(* IEC 61131-3 sources: axftcmlib/src/Axis, 9 files *)

(* ---- Axis.st ---- *)
USING Simatic.Ax.IO.Input;
USING System.Timer;
USING Simatic.Ax.SimpleControlModules;

NAMESPACE Simatic.Ax.axftcmlib
    TYPE INTERNAL
        StatesHoming : (Idle, MoveOutOfSensor, FindReferenceSensor, Done) := Idle;
    END_TYPE

    TYPE INTERNAL
        StateMoveAbsolute : (Idle, Moving, Stopping, Done) := Idle;
    END_TYPE

    TYPE INTERNAL
        MotionMode : (Stopped, Homing, MoveAbsolute, MoveRelative, MoveVelocity);
    END_TYPE

    TYPE
        PlcOpenState : (Ready, Busy, Done, Error) := Ready;
    END_TYPE

    ///Class contains all functions necessary for realisng a motion axis
    ///The motor is used for "powering" the axis
    ///The encoder is needed to monitor the current position
    CLASS Axis
        IMPLEMENTS IAxis
        VAR PUBLIC
            Motor : IMotor;
            Encoder : IEncoder;
            ReferenceSwitch : IBinSignal;
        END_VAR
        VAR PROTECTED
            _stateHoming : StatesHoming;
            _stateMoveAbsolute : StateMoveAbsolute;
            _motionMode : MotionMode;
            _velocity : LREAL;
            _direction : Direction;
            _position : LINT;
            _distance : LINT;
            _plcOpenState : PlcOpenState;
            _done : BOOL;
            _isHomed : BOOL;
            _statusRefSwitch : BOOL;
        END_VAR

        ///Outputs the current status of the axis and executes the protected methods(must be called in every cicle)
        METHOD PUBLIC RunCyclic
            _statusRefSwitch := ReferenceSwitch.Q();
            CASE _motionMode OF
                MotionMode#Stopped:
                    _plcOpenState := PlcOpenState#Ready;
                    ;
                MotionMode#Homing:
                    _plcOpenState := PlcOpenState#Busy;
                    _done := THIS._homing(velocity := _velocity, direction := _direction);
                    IF _done THEN
                        _plcOpenState := PlcOpenState#Done;
                        _isHomed := TRUE;
                        _motionMode := MotionMode#Stopped;
                    END_IF;
                MotionMode#MoveAbsolute:
                    IF (NOT (_isHomed)) THEN
                        _plcOpenState := PlcOpenState#Error;
                        RETURN;
                    END_IF;
                    _plcOpenState := PlcOpenState#Busy;
                    _done := THIS._moveAbsolute(velocity := _velocity, posititon := _position);
                    IF _done THEN
                        _plcOpenState := PlcOpenState#Done;
                        _motionMode := MotionMode#Stopped;
                    END_IF;
                    ;
                MotionMode#MoveRelative:
                    IF (NOT (_isHomed)) THEN
                        _plcOpenState := PlcOpenState#Error;
                        RETURN;
                    END_IF;
                    _plcOpenState := PlcOpenState#Busy;
                    _done := THIS._moveRelative(velocity := _velocity, distance := _distance);
                    IF _done THEN
                        _plcOpenState := PlcOpenState#Done;
                        _motionMode := MotionMode#Stopped;
                    END_IF;
                    ;
                MotionMode#MoveVelocity:
                    _plcOpenState := PlcOpenState#Busy;
                    Motor.Move(_velocity, _direction);

            END_CASE;
        END_METHOD

        ///Moves axis with a velocity
        /// Has to be stopped manually with Halt()
        METHOD PUBLIC MoveVelocity
            VAR_INPUT
                velocity : LREAL;
                direction : Direction;
            END_VAR
            _velocity := velocity;
             _direction := direction;
            _motionMode := MotionMode#MoveVelocity;
        END_METHOD

        ///Moves axis to a new position based on the current position
        METHOD PUBLIC MoveRelative : BOOL
            VAR_INPUT
                velocity : LREAL;
                distance : LINT;
            END_VAR
            _velocity := velocity;
            _distance := distance;
            _motionMode := MotionMode#MoveRelative;
        END_METHOD

        ///Moves axis to a new position based on the default position
        ///homing the axis beforehand is needed to execute this function
        METHOD PUBLIC MoveAbsolute : BOOL
            VAR_INPUT
                velocity : LREAL;
                position : LINT;
            END_VAR
            _velocity := velocity;
            _position := position;
            _motionMode := MotionMode#MoveAbsolute;
        END_METHOD

        ///Moves axis to the default "homing" position (needed for moveAbsolute())
        METHOD PUBLIC Homing : BOOL
            VAR_INPUT
                velocity : LREAL;
                direction : Direction;
            END_VAR
            _velocity := velocity;
            _direction := direction;
            _motionMode := MotionMode#Homing;
        END_METHOD

        ///Homes axis without moving it into default position
        ///Sets position to given value
        METHOD PUBLIC Homing : BOOL
            VAR_INPUT
                Position : LINT;
            END_VAR
            Encoder.SetValue(value := Position);
            _stateHoming := StatesHoming#Done;
            _plcOpenState := PlcOpenState#Done;
            _isHomed := TRUE;
        END_METHOD

        ///Stops movement of the axis
        ///needs to be called manually for MoveVelocity()
        METHOD PUBLIC Halt
            Motor.Halt();
            _motionMode := MotionMode#Stopped;
            _plcOpenState := PlcOpenState#Done;
        END_METHOD
        ///Checks whether the axis is homed or not
        METHOD PUBLIC IsHomed : BOOL
            IsHomed := _isHomed;
        END_METHOD

       //Protected methods are executed by RunCyclic()

       ///Moves axis with a velocity
        /// Has to be stopped manually with Halt()
        METHOD PROTECTED _moveVelocity
            VAR_INPUT
                velocity : LREAL;
                direction : Direction;
            END_VAR
            Motor.Move(velocity, direction);
        END_METHOD

        ///Moves axis to a new position based on the current position
        METHOD PROTECTED _moveRelative : BOOL
            VAR_INPUT
                velocity : LREAL;
                distance : LINT;
            END_VAR
            _moveRelative := THIS._moveAbsolute(velocity := velocity, posititon := Encoder.GetValue() + distance);
        END_METHOD

        ///Moves axis to a new position based on the default position
        ///homing the axis beforehand is needed to execute this function
        METHOD PROTECTED _moveAbsolute : BOOL
            VAR_INPUT
                velocity : LREAL;
                posititon : LINT;
            END_VAR
            VAR_TEMP
                dir : Direction;
            END_VAR
            CASE _stateMoveAbsolute OF
                StateMoveAbsolute#Idle:
                    IF (posititon = Encoder.GetValue()) THEN
                        _stateMoveAbsolute := StateMoveAbsolute#Done;
                        _moveAbsolute := TRUE;
                        Motor.Halt();
                    ELSE
                        _stateMoveAbsolute := StateMoveAbsolute#Moving;
                        Motor.Move(velocity, dir);
                    END_IF;
                    StateMoveAbsolute#Moving:
                    dir := THIS.DecideDirection(enc := Encoder, setPoint := posititon);
                    Motor.Move(velocity, dir);
                    IF (Encoder.GetValue() = posititon) THEN
                        _stateMoveAbsolute := StateMoveAbsolute#Done;
                        Motor.Halt();
                    END_IF;
                    StateMoveAbsolute#Done:
                    _moveAbsolute := TRUE;
                    _stateMoveAbsolute := StateMoveAbsolute#Idle;
                    ;
            END_CASE;
        END_METHOD

        ///Homes axis without moving it into default position
        ///Sets position to given value
        METHOD PROTECTED _homing : BOOL
            VAR_INPUT
                velocity : LREAL;
                direction : Direction;
            END_VAR
            // Reference switch already reached
            // Move out from the Reference switch in opposit direction
            CASE _stateHoming OF
                StatesHoming#Idle:
                    _isHomed := FALSE;
                    IF (ReferenceSwitch.Q()) THEN
                        _stateHoming := StatesHoming#MoveOutOfSensor;
                    ELSE
                        _stateHoming := StatesHoming#FindReferenceSensor;
                    END_IF;
                StatesHoming#MoveOutOfSensor:
                    Motor.Move(direction := THIS._oppositDirection(direction := direction));
                    IF (ReferenceSwitch.QFal()) THEN
                        Motor.Halt();
                        _stateHoming := StatesHoming#FindReferenceSensor;
                    END_IF;
                StatesHoming#FindReferenceSensor:
                    Motor.Move(direction := direction);
                    IF (ReferenceSwitch.QRis()) THEN
                        Motor.Halt();
                        Encoder.SetValue(value := 0);
                        _stateHoming := StatesHoming#Done;
                    END_IF;
                StatesHoming#Done:
                    _homing := TRUE;
                    _stateHoming := StatesHoming#Idle;
            END_CASE;
            ;
        END_METHOD

        ///inverts the current direction
        METHOD PROTECTED _oppositDirection : Direction
            VAR_INPUT
                direction : Direction;
            END_VAR
            IF (direction = Direction#Forward) THEN
                _oppositDirection := Direction#Reverse;
            ELSE
                _oppositDirection := Direction#Forward;
            END_IF;
        END_METHOD

        ///decides the needed direction to reach setpoint
        METHOD PROTECTED DecideDirection : Direction
            VAR_INPUT
                enc : IEncoder;
                setpoint : LINT;
            END_VAR
            IF (setpoint >= enc.GetValue()) THEN
                DecideDirection := Direction#Forward;
            ELSE
                DecideDirection := Direction#Reverse;
            END_IF;
        END_METHOD

        ///Outputs current status of the PLC
        METHOD PUBLIC GetPlcOpenState : PlcOpenState
            GetPlcOpenState := _plcOpenState;
        END_METHOD
        ///Returns whether the axis is busy with a movement command
        METHOD PUBLIC IsRunning : BOOL
            IsRunning := _plcOpenState = PlcOpenstate#Busy;
        END_METHOD
    END_CLASS

END_NAMESPACE

(* ---- IAxis.st ---- *)
NAMESPACE Simatic.Ax.axftcmlib

    TYPE
        Direction : (Forward, Reverse, Undefined) := Forward;
    END_TYPE

    ///Interface for implementing an axis
    ///Contains basic functions needed for realising an axis
    INTERFACE IAxis
        ///Moves axis wit given velcity in a given direction
        METHOD MoveVelocity
            VAR_INPUT
                velocity : LREAL;
                direction : Direction;
            END_VAR
        END_METHOD
        ///Moves axis to destination based on current position
        METHOD MoveRelative : BOOL
            VAR_INPUT
                velocity : LREAL;
                distance : LINT;
            END_VAR
        END_METHOD
        ///Moves axis to a new position based on the default position
        METHOD MoveAbsolute : BOOL
            VAR_INPUT
                velocity : LREAL;
                position : LINT;
            END_VAR
        END_METHOD
        ///Stops axis
        METHOD Halt
        END_METHOD
        ///Moves axis into the default position
        METHOD Homing : BOOL
            VAR_INPUT
                velocity : LREAL;
                direction : Direction;
            END_VAR
        END_METHOD
        ///Resets current position to deafult value without actual movement
        METHOD Homing : BOOL
            VAR_INPUT
                Position : LINT;
            END_VAR
        END_METHOD
        ///Returns whether the defaultposition is set
        METHOD IsHomed : BOOL
        END_METHOD
        ///Returns whether the axis is busy with a movement command
        METHOD IsRunning : BOOL
        END_METHOD
    END_INTERFACE

END_NAMESPACE

(* ---- IMotor.st ---- *)
NAMESPACE Simatic.Ax.axftcmlib
    INTERFACE IMotor
        METHOD Move
            VAR_INPUT
                velocity : LREAL;
                direction : Direction;
            END_VAR
        END_METHOD
        METHOD Halt
        END_METHOD
    END_INTERFACE
END_NAMESPACE

(* ---- ITimeprovider.st ---- *)
USING Siemens.Simatic.S71500.Clocks;
NAMESPACE Simatic.Ax.axftcmlib

    INTERFACE ITimeprovider
        Method GetElapsedSeconds :LREAL
        END_METHOD
    END_INTERFACE

    CLASS TimeProvider Implements ITimeprovider

    VAR
     _measurement : RuntimeMeasurement;
     _timeOfOperations : LTIME;
    END_VAR

    METHOD PUBLIC GetElapsedSeconds : LREAL
            _timeOfOperations := _measurement.Stop();
            GetElapsedSeconds := _measurement.GetElapsedSeconds();//time passed in seconds
            _measurement.Start();
    END_METHOD

    END_CLASS

    CLASS TimeProviderMOCK_100ms_const Implements ITimeprovider

        VAR
         _measurement : RuntimeMeasurement;
         _timeOfOperations : LTIME;
        END_VAR

        METHOD PUBLIC GetElapsedSeconds : LREAL
              GetElapsedSeconds := 0.1;
        END_METHOD

        END_CLASS

END_NAMESPACE

(* ---- AxisBase.st ---- *)
USING Simatic.Ax.Commands;

NAMESPACE Simatic.Ax.axftcmlib.Motion

    CLASS INTERNAL ABSTRACT AxisBase IMPLEMENTS itfAxis
        VAR PROTECTED
            _AxisRef : REF_TO TO_Axis;
        END_VAR

        METHOD PROTECTED ABSTRACT MakeAxisAbstract END_METHOD

        METHOD PUBLIC Attach
            VAR_INPUT
                axis : REF_TO TO_Axis;
            END_VAR
            _AxisRef := axis;
        END_METHOD

        METHOD PROTECTED IsAttached : BOOL
            IsAttached := _AxisRef <> NULL;
        END_METHOD

        METHOD PUBLIC PowerOn
            _AxisRef^.isPowerdOn := TRUE;
        END_METHOD

        METHOD PUBLIC PowerOff
            _AxisRef^.isPowerdOn := FALSE;
        END_METHOD

    END_CLASS

END_NAMESPACE

(* ---- Motor.st ---- *)
USING Simatic.Ax.IO.Output;
USING Simatic.Ax.axftcmlib;

NAMESPACE Simatic.Ax.axftcmlib

    CLASS MotorFT
        IMPLEMENTS IMotor
        VAR PUBLIC
            Forward : IBinOutput;
            Reverse : IBinOutput;
        END_VAR
        VAR PROTECTED
        END_VAR
        METHOD PUBLIC Move
            VAR_INPUT
                velocity : LREAL;
                direction : Direction;
            END_VAR
            IF (direction = Direction#Forward) THEN
                Forward.SetOn();
                Reverse.SetOff();
            ELSE
                Reverse.SetOn();
                Forward.SetOff();
            END_IF;
            ;
        END_METHOD
        METHOD PUBLIC Halt
            Reverse.SetOff();
            Forward.SetOff();
            ;
        END_METHOD
    END_CLASS

END_NAMESPACE

(* ---- PLCOpentateGuard.st ---- *)
USING Simatic.Ax.StateFramework;
NAMESPACE Simatic.Ax.axftcmlib
    // CLASS PLCOpenstateGuard IMPLEMENTS IGuard

    //     VAR PUBLIC
    //         UsedAxis : REF_TO AXIS;
    //     END_VAR

    //     VAR
    //         CurrentState : PlcOpenState;
    //     END_VAR

    //     METHOD PUBLIC Check : BOOL
    //         CurrentState := UsedAxis^.GetPlcOpenState();
    //        IF CurrentState = PlcOpenState#DONE THEN
    //         Check := TRUE;
    //        ELSE
    //         Check := FALSE;
    //        END_IF;
    //     END_METHOD

    //     METHOD PUBLIC Reset
    //         ;
    //     END_METHOD

    // END_CLASS
    CLASS PLCOpenstateGuard IMPLEMENTS IGuard
        VAR PUBLIC
            Axis : REF_TO Axis;
        END_VAR

        METHOD PUBLIC Check : BOOL
            Check := (Axis^.GetPlcOpenState() = PlcOpenState#Done);
        END_METHOD

        METHOD PUBLIC Reset
            ;
        END_METHOD
    END_CLASS
END_NAMESPACE

(* ---- TimeBasedEncoder.st ---- *)
USING Simatic.Ax.SimpleControlModules;
USING Simatic.Ax.IO.Output;
USING Simatic.Ax.IO.Input;

USING System.Timer;

NAMESPACE Simatic.Ax.axftcmlib
    CLASS TimeBasedEncoder Implements IEncoder
        VAR PUBLIC
            Velocity : LREAL; // m/s
            EncoderAxis : IAxis;
            TimeProvider : ITimeprovider;
            //--------------------------
            RealPosition : LREAL;
        END_VAR

        VAR PROTECTED
            _position : LREAL; // mm
        END_VAR

        /// Reset encoder position to zero
        METHOD PUBLIC Reset
            _position := 0.0;
        END_METHOD

        /// Set encoder to specific position
        /// value : Position which is set
        METHOD PUBLIC SetValue
            VAR_INPUT
                value : LINT;
            END_VAR
            _position := TO_LREAL(value);
        END_METHOD

        /// Returns the actual encoder position
        /// Actual encoder position
        METHOD PUBLIC GetValue : LINT
            GetValue := TO_LINT(_position);
            RealPosition := _position;
        END_METHOD

        /// Evaluate encoder signals
        METHOD PUBLIC Evaluate
            VAR_TEMP
             ds : LREAL;
             dt : LREAL;
            END_VAR

            dt := TimeProvider.GetElapsedSeconds();//time passed in seconds
            ds := Velocity * dt;
            IF (EncoderAxis.IsRunning()) THEN //If Axis is running
                _position := _position + ds;
            END_IF;
        END_METHOD
        //=========================================================
        /// Returns if the encoder has moved
        /// Encoder has moved
        METHOD PUBLIC HasMoved : BOOL
            // HasMoved := _encoderHasMoved;
            // _encoderHasMoved := FALSE;
           ;
        END_METHOD

        /// Counts the relative pulses since the last Reset or ResetRelative command
        METHOD PUBLIC RelativeCount : LINT
            //RelativeCount := _encoderRelativeCounter.CounterValue() MOD Modulo;
            ;
        END_METHOD

        /// Reset the relative counter
        METHOD PUBLIC ResetRelative
            //_encoderRelativeCounter.SetCounterValue(LINT#0);
           ;
        END_METHOD

        METHOD PUBLIC SetDirection
            VAR_INPUT
                mode : CountMode;
            END_VAR
            ;
        END_METHOD

        METHOD PUBLIC GetModulo : LINT
          ;
        END_METHOD
    END_CLASS
    END_NAMESPACE

(* ---- Timeprovider.st ---- *)
USING Siemens.Simatic.S71500.Clocks;
 NAMESPACE Simatic.Ax.axftcmlib
    /// Timeprovider based on RuntimeMeasurement
    CLASS TimeProvider
        IMPLEMENTS ITimeprovider
        VAR
            _measurement : RuntimeMeasurement;
            _elapsedTimeInSeconds : LREAL;
        END_VAR

        // mus be called in every cycle
        METHOD PUBLIC Evaluate
            _measurement.Stop();
         _elapsedTimeInSeconds := _measurement.GetElapsedSeconds(); //time passed in seconds
         _measurement.Start();
       END_METHOD

     METHOD PUBLIC GetElapsedSeconds : LREAL
        GetElapsedSeconds := _elapsedTimeInSeconds;
     END_METHOD
    END_CLASS

    /// Mock for a ITimePrivider wich returns always 100ms.
    CLASS TimeProviderMOCK_100ms_const
        IMPLEMENTS ITimeprovider

        METHOD PUBLIC GetElapsedSeconds : LREAL
         GetElapsedSeconds := 0.1;
        END_METHOD
    END_CLASS
END_NAMESPACE
